TYPE generatedOrderStatusWord_TypeStruct :
STRUCT
	

	knifeOutOfRangeArr			: ARRAY [1..5] OF BOOL;
	scorerOutOfRangeArr		: ARRAY [1..8] OF BOOL;


	orderNotOk				: BOOL;	


END_STRUCT
END_TYPE

(* stored: Version 1.1.0.1
   DUT generatedOrderStatusWord_TypeStruct: Id {66789238-01e2-45fc-83fa-d4546d93cfef} *)
